FUNCTION_BLOCK SWITCH (* Switch(demultiplex)an event *)
  (* Standard: 61499-1; Classification: Event Processing; Function: Event Switch *)
  (* Version 7.0, 01/12/2011, LAPAS, UDESC *)
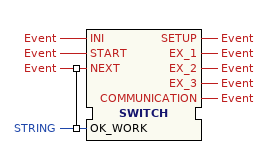
  EVENT_INPUT
    INI; (* Inicializa o bloco *)
    START; (* Inicia o primeiro evento de saida *)
    NEXT WITH OK_WORK; (* Gera o proximo evento de saida *)
  END_EVENT
  EVENT_OUTPUT
    SETUP; (* Setup da maquina *)
    EX_1; (* Executable 1 *)
    EX_2; (* Executable 2 *)
    EX_3; (* Executable 3 *)
    COMMUNICATION; (* comunicacao *)
  END_EVENT
  VAR_INPUT
    OK_WORK : STRING;
  END_VAR
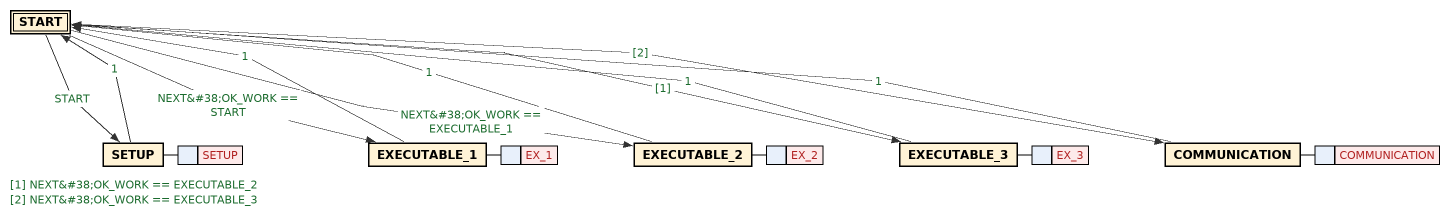
  EC_STATES
    START;
    SETUP : -> SETUP;
    EXECUTABLE_1 : -> EX_1;
    EXECUTABLE_2 : -> EX_2;
    EXECUTABLE_3 : -> EX_3;
    COMMUNICATION : -> COMMUNICATION;
  END_STATES
  EC_TRANSITIONS
    START TO SETUP := START;
    START TO EXECUTABLE_1 := NEXT&#38;OK_WORK == START;
    START TO EXECUTABLE_2 := NEXT&#38;OK_WORK == EXECUTABLE_1;
    START TO EXECUTABLE_3 := NEXT&#38;OK_WORK == EXECUTABLE_2;
    START TO COMMUNICATION := NEXT&#38;OK_WORK == EXECUTABLE_3;
    SETUP TO START := 1;
    EXECUTABLE_1 TO START := 1;
    EXECUTABLE_2 TO START := 1;
    EXECUTABLE_3 TO START := 1;
    COMMUNICATION TO START := 1;
  END_TRANSITIONS
END_FUNCTION_BLOCK
